// TIA Portal V18 export
// export: Created 2026-06-05T07:40:25.1259938Z, ExportSetting WithDefaults, DisplayName Totally Integrated Automation Portal, DisplayVersion V18, DisplayName TIA Portal Openness, DisplayVersion V18, DisplayName TIA Portal Version Control Interface, DisplayVersion V18, DisplayName STEP 7 Professional, DisplayVersion V18, DisplayName STEP 7 Safety, DisplayVersion V18, DisplayName WinCC Professional, DisplayVersion V18
ORGANIZATION_BLOCK "Main"   // OB1, LAD, ProgramCycle
TITLE = "Main Program Sweep (Cycle)"
{ S7_Optimized_Access := 'TRUE' }
VERSION : 0.1
// stored: AutoNumber true, IsIECCheckEnabled false, SetENOAutomatically false
   VAR_INPUT
      Initial_Call : Bool;   // Initial call of this OB
      Remanence : Bool;   // =True, if remanent data are available
   END_VAR
BEGIN

REGION Network 1: Call FC_PLC1_Logic
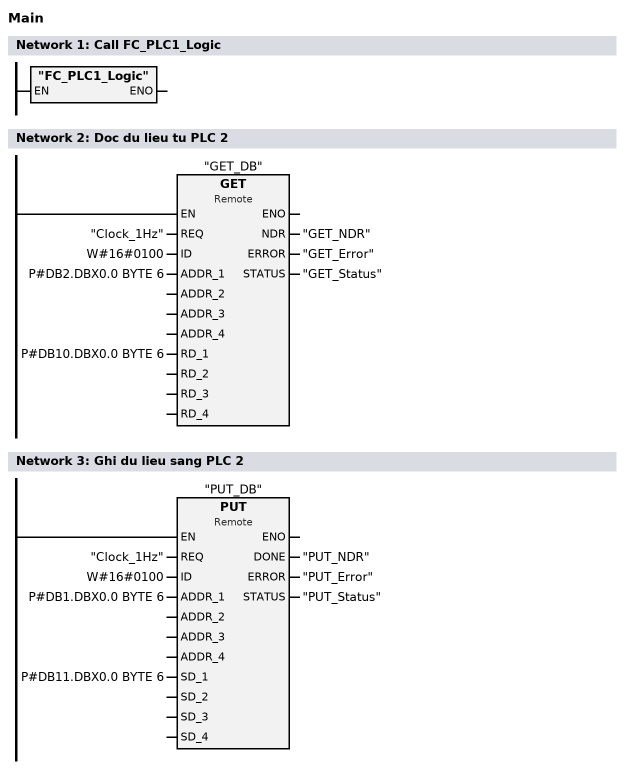
   RUNG wire#powerrail
      "FC_PLC1_Logic"()
   END_RUNG
   // the same network as SCL:
   "FC_PLC1_Logic"();
END_REGION

REGION Network 2: Doc du lieu tu PLC 2
   RUNG wire#powerrail
      { S7_Templates := "[remote_type := Remote, local_type := Variant]" } "GET_DB".GET(REQ := "Clock_1Hz", ID := W#16#0100, ADDR_1 := P#DB2.DBX0.0 BYTE 6, ADDR_2 :=, ADDR_3 :=, ADDR_4 :=, RD_1 := P#DB10.DBX0.0 BYTE 6, RD_2 :=, RD_3 :=, RD_4 :=, NDR => "GET_NDR", ERROR => "GET_Error", STATUS => "GET_Status")
   END_RUNG
   // the same network as SCL:
   "GET_DB"(REQ := "Clock_1Hz",   // GET
            ID := W#16#0100,
            ADDR_1 := P#DB2.DBX0.0 BYTE 6,
            RD_1 := P#DB10.DBX0.0 BYTE 6,
            NDR => "GET_NDR",
            ERROR => "GET_Error",
            STATUS => "GET_Status");
END_REGION

REGION Network 3: Ghi du lieu sang PLC 2
   RUNG wire#powerrail
      { S7_Templates := "[remote_type := Remote, local_type := Variant]" } "PUT_DB".PUT(REQ := "Clock_1Hz", ID := W#16#0100, ADDR_1 := P#DB1.DBX0.0 BYTE 6, ADDR_2 :=, ADDR_3 :=, ADDR_4 :=, SD_1 := P#DB11.DBX0.0 BYTE 6, SD_2 :=, SD_3 :=, SD_4 :=, DONE => "PUT_NDR", ERROR => "PUT_Error", STATUS => "PUT_Status")
   END_RUNG
   // the same network as SCL:
   "PUT_DB"(REQ := "Clock_1Hz",   // PUT
            ID := W#16#0100,
            ADDR_1 := P#DB1.DBX0.0 BYTE 6,
            SD_1 := P#DB11.DBX0.0 BYTE 6,
            DONE => "PUT_NDR",
            ERROR => "PUT_Error",
            STATUS => "PUT_Status");
END_REGION
END_ORGANIZATION_BLOCK
